Universal Robots PolyScope program: adaptiveGripper.urp

Program adaptiveGripper (installation=20240827 directory=/programs/Demos/water createdIn=5.15.1 lastSavedIn=5.15.1 robotSerialNumber=20245500285)
Calibrated DH parameters: a=[0.000097, -0.210459, -0.026602, 0.000137, 0.000078, 0]; d=[0.162601, 254.180657, -54.076236, -199.970743, 0.099615, 0.099684]; alpha=[1.569796, -0.001455, 0.001957, 1.570525, -1.571561, 0]; deltaTheta=[0, -1.053331, 8.839472, -1.50296, 0.000002, 0]
InitVariablesNode
Robot Program (runOnlyOnce=false)
  Script: usb = rpc_factory("xmlrpc","http://192.168.1.7:9120/RPC2")
  counter := 0
  Loop Forever
    Script: usb.open()
    SuppressedNode
      Wait Sleep waitTime=0.5
    Popup Message (haltProgram=false message=12 inputType=Text)
    SuppressedNode
      MoveJ speed 60 deg/s, acceleration 80 deg/s^2 (useActiveTCP=true) feature=Base
        SuppressedNode
          Waypoint 路点_1: TCP in base x=191.611 y=-565.461 z=6.817 mm, rx=-2.2765 ry=-2.1528 rz=-0.0082 rad; joints [95.723, -64.864, 103.956, -128.576, -90.128, 99.099] deg; TCP offset x=-0.17 y=0 z=192.95 mm, rx=0 ry=0 rz=0 rad
    Script: usb.adaptiveClose()
    SuppressedNode
      Wait Sleep waitTime=0.5
    SuppressedNode
      MoveL speed 250 mm/s, acceleration 1200 mm/s^2 (useActiveTCP=true) feature=Base
        Waypoint 路点_2: TCP in base x=191.566 y=-565.44 z=47.246 mm, rx=-2.2766 ry=-2.1527 rz=-0.0083 rad; joints [95.72, -68.174, 101.706, -123.011, -90.114, 99.104] deg
    SuppressedNode
      MoveJ speed 60 deg/s, acceleration 80 deg/s^2 (useActiveTCP=true) feature=Base
        Waypoint 路点_1: TCP in base x=191.611 y=-565.461 z=6.817 mm, rx=-2.2765 ry=-2.1528 rz=-0.0082 rad; joints [95.723, -64.864, 103.956, -128.576, -90.128, 99.099] deg
    Popup Message (haltProgram=false message=12 inputType=Text)
    Script: counter=counter+1
